FUNCTION_BLOCK ABSTRACT FB_ApplicationConfigRoot
VAR
	_LinkVariableManager : FB_LinkVariableManager;
	_ReferenceManager : FB_ReferenceManager;
	_ModuleTypeRegistry : FB_ModuleTypeRegistry;
	_ModuleConfigurationManager : FB_ModuleConfigurationManager;
	_bRegistrationAttempted : BOOL;
	_bRegistered : BOOL;
	_bError : BOOL;
	_hrErrorCode : HRESULT;
	_sErrorMessage : STRING(255);
END_VAR

PROPERTY PUBLIC FINAL Busy : BOOL
GET
Busy := _bRegistered AND NOT _bError AND _ModuleConfigurationManager.Busy;
END_GET
END_PROPERTY

PROPERTY PUBLIC FINAL Error : BOOL
GET
Error := _bError;
END_GET
END_PROPERTY

PROPERTY PUBLIC FINAL ErrorCode : HRESULT
GET
ErrorCode := _hrErrorCode;
END_GET
END_PROPERTY

PROPERTY PUBLIC FINAL ErrorMessage : STRING(255)
GET
ErrorMessage := _sErrorMessage;
END_GET
END_PROPERTY

METHOD PROTECTED H_RegisterBaseUnits
END_METHOD

METHOD PROTECTED H_RegisterIo
END_METHOD

METHOD PROTECTED H_RegisterModuleTypes
END_METHOD

METHOD PROTECTED H_RunModules
VAR_INPUT
	VariableNodeReader : I_VariableNodeReader;
END_VAR
VAR_IN_OUT CONSTANT
	SystemContext : ST_SystemContext;
END_VAR
END_METHOD

METHOD PUBLIC FINAL M_CyclicInput
IF Ready THEN
	_LinkVariableManager.M_CyclicInput();
END_IF
END_METHOD

METHOD PUBLIC FINAL M_CyclicModules
VAR_IN_OUT CONSTANT
	SystemContext : ST_SystemContext;
END_VAR
IF Ready THEN
	H_RunModules(
		SystemContext := SystemContext,
		VariableNodeReader := _LinkVariableManager);
END_IF
END_METHOD

METHOD PUBLIC FINAL M_CyclicOutput
IF Ready THEN
	_LinkVariableManager.M_CyclicOutput();
END_IF
END_METHOD

METHOD PUBLIC FINAL M_PollConfiguration
VAR
	bRegistrationSessionStarted : BOOL;
	bRegistrationSealed : BOOL;
END_VAR
IF NOT _bRegistrationAttempted THEN
	_bRegistrationAttempted := TRUE;

	// The base class owns the Infrastructure registration session.
	bRegistrationSessionStarted := _LinkVariableManager.M_BeginInfrastructureRegistration();
	IF NOT bRegistrationSessionStarted THEN
		M_SetError(
			Message := _LinkVariableManager.ErrorMessage,
			ErrorCode := 0);
	ELSE
		H_RegisterIo();

		// Always seal an opened session. On a registration error this also rolls
		// back every Infrastructure node declared during this attempt.
		bRegistrationSealed := _LinkVariableManager.M_SealInfrastructureRegistration();
		IF NOT bRegistrationSealed THEN
			M_SetError(
				Message := _LinkVariableManager.ErrorMessage,
				ErrorCode := 0);
		END_IF
	END_IF

	IF NOT _bError THEN
		H_RegisterBaseUnits();
	END_IF
	IF NOT _bError THEN
		H_RegisterModuleTypes();
	END_IF

	_bRegistered := NOT _bError;
END_IF

IF NOT _bRegistered OR _bError THEN
	RETURN;
END_IF

_ModuleConfigurationManager(
	Execute := TRUE,
	FilePath := Param_Config.ModuleConfigFilePath,
	LinkVariableManager := _LinkVariableManager,
	ReferenceManager := _ReferenceManager,
	ModuleTypeRegistry := _ModuleTypeRegistry);

IF _ModuleConfigurationManager.Error THEN
	M_SetError(
		Message := _ModuleConfigurationManager.ErrorMessage,
		ErrorCode := _ModuleConfigurationManager.ErrorCode);
END_IF
END_METHOD

METHOD PROTECTED FINAL M_RegisterBaseUnit : BOOL
VAR_INPUT
	BaseUnit : I_BaseUnit;
END_VAR
M_RegisterBaseUnit := FALSE;
IF _bError THEN
	RETURN;
END_IF

M_RegisterBaseUnit := _ReferenceManager.M_RegisterReference(BaseUnit := BaseUnit);
IF NOT M_RegisterBaseUnit THEN
	M_SetError(
		Message := _ReferenceManager.ErrorMessage,
		ErrorCode := 0);
END_IF
END_METHOD

METHOD PROTECTED FINAL M_RegisterIoNode : BOOL
VAR_INPUT
	Variable : ANY;
	Access : E_VariableAccess;
END_VAR
M_RegisterIoNode := FALSE;
IF _bError THEN
	RETURN;
END_IF

M_RegisterIoNode := _LinkVariableManager.M_RegisterInfrastructureNode(
	Variable := Variable,
	Access := Access);
IF NOT M_RegisterIoNode THEN
	M_SetError(
		Message := _LinkVariableManager.ErrorMessage,
		ErrorCode := 0);
END_IF
END_METHOD

METHOD PROTECTED FINAL M_RegisterModuleType : BOOL
VAR_INPUT
	ModuleTypeName : T_ModuleTypeName;
	Adapter : I_ModuleConfigurationAdapter;
END_VAR
M_RegisterModuleType := FALSE;
IF _bError THEN
	RETURN;
END_IF

M_RegisterModuleType := _ModuleTypeRegistry.M_Register(
	ModuleTypeName := ModuleTypeName,
	Adapter := Adapter);
IF NOT M_RegisterModuleType THEN
	M_SetError(
		Message := _ModuleTypeRegistry.ErrorMessage,
		ErrorCode := 0);
END_IF
END_METHOD

METHOD PRIVATE M_SetError
VAR_INPUT
	Message : STRING(255);
	ErrorCode : HRESULT;
END_VAR
IF NOT _bError THEN
	_bError := TRUE;
	_hrErrorCode := ErrorCode;
	IF Message = '' THEN
		_sErrorMessage := 'Application configuration initialization failed.';
	ELSE
		_sErrorMessage := Message;
	END_IF
END_IF
END_METHOD

PROPERTY PUBLIC FINAL Ready : BOOL
GET
Ready := _bRegistered AND NOT _bError AND _ModuleConfigurationManager.Ready;
END_GET
END_PROPERTY

END_FUNCTION_BLOCK

(* stored: Version 1.1.0.1, ProductVersion 3.1.4026.18
   POU FB_ApplicationConfigRoot: Id {ac023e93-0e8c-4841-9092-5acf2380946d}, SpecialFunc None
   Folder Hook Method: Id {36eef1a3-3ffe-4697-afea-6d6c4afaf709}
   Property Busy: Id {92192890-fd81-4d3b-9bea-ca078aa01c09}
   Get Get: Id {43c4e7f2-3690-429f-a433-7d60e1316c5c}
   Property Error: Id {948f0dda-5a32-41b8-b963-ec63c7a801e9}
   Get Get: Id {22ad876d-8540-456c-a6e9-8eede70a7eb5}
   Property ErrorCode: Id {0889f68d-3e5f-4161-ad59-544a8a8bfdab}
   Get Get: Id {8d802ab3-d105-4e20-8583-2cef7d00b43f}
   Property ErrorMessage: Id {031b9a1c-934b-488e-87d8-d824b0526ca4}
   Get Get: Id {aacab3bd-a53f-44c0-9dbd-e0758a727ce1}
   Method H_RegisterBaseUnits: Id {d75fd37d-b59c-48ec-8ca8-3b1db41eb01a}
   Method H_RegisterIo: Id {e1e2f45f-84f1-49a2-af6e-e2551f0bdaac}
   Method H_RegisterModuleTypes: Id {c08dab9f-dbd2-46bf-ab82-4ee25f82d6a9}
   Method H_RunModules: Id {c9048f6b-9da6-4292-8e8f-f3456e44a81c}
   Method M_CyclicInput: Id {bdd61f85-631c-46ea-9b9e-021c6badf010}
   Method M_CyclicModules: Id {efe30913-6738-4a2f-8f94-a3174c6941c4}
   Method M_CyclicOutput: Id {edeb8ca1-72ab-4bc5-85a0-c9f83942239b}
   Method M_PollConfiguration: Id {3afd629d-8905-4d8b-9a7e-d84357b3398c}
   Method M_RegisterBaseUnit: Id {88aa0f03-12da-42fb-8adf-a837e6fa3d7d}
   Method M_RegisterIoNode: Id {3de1be0c-87c0-481c-9f44-089699215ef2}
   Method M_RegisterModuleType: Id {0e519d82-3126-4b92-a042-9bee77d06d8a}
   Method M_SetError: Id {bb8fedaf-e4d5-4b3c-ab9f-9246cc78fb7e}
   Property Ready: Id {0b170b93-5657-4b3a-bbd4-34f1f336bea3}
   Get Get: Id {d22bb374-9b62-464a-9439-80e9c5fc1052} *)
